// TwinCAT 3 PLC project PLC
// ProgramVersion: 3.1.4024.0
// libraries:
//   Tc2_CncHli, * (Beckhoff Automation GmbH)
//   Tc2_Standard, * (Beckhoff Automation GmbH)
//   Tc2_System, * (Beckhoff Automation GmbH)
//   Tc3_Module, * (Beckhoff Automation GmbH)
//   Triamec EtherCAT Lib, * (Triamec Motion AG)
// project tree:
//   GVLs/ Triamec_GVL.TcGVL
//   / PlcTask.TcTTO
//   POUs/ CNC_Axis.TcPOU, MAIN.TcPOU
// real-time tasks:
//   TASK PlcTask: cycle T#10ms, priority 20, ADS port 350
// I/O:
//   DEVICE Device 1 (EtherCAT), AmsNetId 10.20.34.98.2.1
//     Drive 1 (TSD) [TSD_minFW4.22]
//       modules: Axis 0, Axis 0, Axis 0, Axis 0, Axis 0, Axis 1, Axis 1, Axis 1, Axis 1, Axis 1
// variable links:
//   CNC/Axes/Axis_1 <-> Device 1 (EtherCAT)/Drive 1 (TSD)
//     Inputs/ActualPosition <-> Axis 0/MainInputs/ActualPosition
//     Inputs/ActualVelocity <-> Axis 0/VelocityInputs/ActualVelocity
//     Inputs/MessageId <-> Axis 0/Diagnostic / Digital Inputs/MessageId
//     Inputs/Mode of Operation Display <-> Axis 0/MainInputs/Mode of Operation Display
//     Inputs/PositionError <-> Axis 0/PositionInputs/PositionError
//     Inputs/Status Word <-> Axis 0/MainInputs/Status Word
//     Inputs/TorqueActual <-> Axis 0/TorqueInputs/TorqueActual
//     Inputs/WcState <-> WcState/WcState
//     Outputs/Auxiliary Byte <-> Axis 0/MainOutputs/Auxiliary Byte
//     Outputs/Control Word <-> Axis 0/MainOutputs/Control Word
//     Outputs/Mode of Operation <-> Axis 0/MainOutputs/Mode of Operation
//     Outputs/TargetPosition <-> Axis 0/PositionOutputs/TargetPosition
//     Outputs/TargetTorque <-> Axis 0/TorqueOutputs/TargetTorque
//     Outputs/TargetVelocity <-> Axis 0/VelocityOutputs/TargetVelocity
//   CNC/Axes/Axis_2 <-> Device 1 (EtherCAT)/Drive 1 (TSD)
//     Inputs/ActualPosition <-> Axis 1/MainInputs/ActualPosition
//     Inputs/ActualVelocity <-> Axis 1/VelocityInputs/ActualVelocity
//     Inputs/MessageId <-> Axis 1/Diagnostic / Digital Inputs/MessageId
//     Inputs/Mode of Operation Display <-> Axis 1/MainInputs/Mode of Operation Display
//     Inputs/PositionError <-> Axis 1/PositionInputs/PositionError
//     Inputs/Status Word <-> Axis 1/MainInputs/Status Word
//     Inputs/TorqueActual <-> Axis 1/TorqueInputs/TorqueActual
//     Inputs/WcState <-> WcState/WcState
//     Outputs/Auxiliary Byte <-> Axis 1/MainOutputs/Auxiliary Byte
//     Outputs/Control Word <-> Axis 1/MainOutputs/Control Word
//     Outputs/Mode of Operation <-> Axis 1/MainOutputs/Mode of Operation
//     Outputs/TargetPosition <-> Axis 1/PositionOutputs/TargetPosition
//     Outputs/TargetTorque <-> Axis 1/TorqueOutputs/TargetTorque
//     Outputs/TargetVelocity <-> Axis 1/VelocityOutputs/TargetVelocity

CONFIGURATION PLC
    RESOURCE PLC ON TwinCAT3
        TASK PlcTask(INTERVAL := T#10ms, PRIORITY := 20);
        PROGRAM MAIN WITH PlcTask : MAIN;
    END_RESOURCE
END_CONFIGURATION

// ---- GVLs/Triamec_GVL.TcGVL
VAR_GLOBAL
	gEnableAxes			: BOOL;	(* variable to enable all axes *)
	gStatusAxesEnabled 	: BOOL;	(* variable indicates that all axes enabled *)	
END_VAR

// ---- POUs/MAIN.TcPOU
PROGRAM MAIN
VAR
	Axis		: ARRAY [0..1] OF CNC_Axis; // CNC axis
	Hli 		: MCV_HliInterface;
	axisIdx		: UINT;
END_VAR

(* configuration *)
Axis[0].config.driveId	:= 1001;				// Drive 1 (TSD)/EtherCAT/EtherCAT-Addr.
Axis[0].config.netId	:= '192.168.10.99.2.1';	// Drive 1 (TSD)^InfoData^AdsAddr^netId
Axis[0].config.axisNumber:= 0;					// first (0) or second (1) axis of a dual axis drive
Axis[0].config.axisId	:= 0;					// cnc-axis-id used in events
Axis[1].config.driveId	:= 1001;				// Drive 1 (TSD)/EtherCAT/EtherCAT-Addr.
Axis[1].config.netId	:= '192.168.10.99.2.1';	// Drive 1 (TSD)^InfoData^AdsAddr^netId
Axis[1].config.axisNumber:= 1;					// first (0) or second (1) axis of a dual axis drive
Axis[1].config.axisId	:= 1;					// cnc-axis-id used in events

(* HLI interface *)
IF NOT Hli.Initialized THEN
	Hli(); //initialize HLI
END_IF

(* Axis handler *)
IF Hli.Initialized THEN
	gStatusAxesEnabled := TRUE;
	FOR axisIdx := 0 TO SIZEOF(Axis)/SIZEOF(Axis[0])-1 DO
		Axis[axisIdx].enable := gEnableAxes;
		Axis[axisIdx]();
		IF NOT Axis[axisIdx].enabled THEN
			gStatusAxesEnabled := FALSE;
		END_IF
	END_FOR
END_IF

END_PROGRAM

// ---- POUs/CNC_Axis.TcPOU
FUNCTION_BLOCK CNC_Axis EXTENDS TE_AxisBase0
VAR_INPUT
	enable		: BOOL;
	hold		: BOOL;
END_VAR
VAR_OUTPUT
	ready		: BOOL;
	enabled		: BOOL;
	referenced	: BOOL;
	state		: DWORD;
	error		: BOOL;
END_VAR
VAR
	pAxis		: POINTER TO HIGH_LEVEL_INTERFACE_AX;
END_VAR

(* Triamec Motion AG, 6340 Baar, Switzerland    *)
(* Sample Code may be adapted to customer needs *)
(* -------------------------------------------- *)
(* 
	we do not want any offset between drive and cnc 
    because the drives have there own setPosition
	therefore set the following parameters in the axis of the cnc:
		kenngr.abs_pos_gueltig			1
		kenngr.set_refpos_mode         	OFFSET
		kenngr.set_refpos_offset		0
	this mode ensures, that the cnc does not set cmdPos=actPos when
	MCControlBoolUnit_SetReferencePosition is set
	
	To enable homing using G74 set the following in every axis configuration
	kenngr.device_id  8             ( turn off the target reached check before homing)
*)

IF config.axisId >= 0 AND HLI_SYS_AX_MAXIDX > config.axisId THEN (* check for axis id *)
	(* be careful, array indices start with 0 in TwinCAT 3. Axis starts with 1 *)
	pAxis := gpAx[config.axisId];
	pAxis^.head.plc_present_w := TRUE;
	
	(* enable PLC to drive HLI interface *)
	pAxis^.lr_mc_control.torque_permission.enable_w			:= TRUE;
	pAxis^.lr_mc_control.release_feedhold.enable_w 			:= TRUE;
	pAxis^.lr_mc_control.drive_on.enable_w 					:= TRUE;		
	(* set reference postion offset *)
//	pAxis^.lr_mc_control.set_reference_position.enable_w	:= TRUE;
	(* enable the axis to tracking operation (follow up) *)
	pAxis^.lr_mc_control.follow_up.enable_w 				:= TRUE;

	(* set regulation and feed *)
	pAxis^.lr_mc_control.torque_permission.command_w		:= enable;
	pAxis^.lr_mc_control.release_feedhold.command_w 		:= NOT Hold;
	pAxis^.lr_mc_control.drive_on.command_w 				:= TRUE;
	
	state := pAxis^.lr_state.native_drive_state_r;
	error := (state AND 16#8) <> 0;
	
	(* The axis is set to tracking operation (follow up) on or off, i.e. the control loop is opened.
	   The command position implicitly is set to the actual position. *)
	pAxis^.lr_mc_control.follow_up.command_w				:= (state AND 16#0100) <> 0;
	(* HomingPosition *)
//	pAxis^.lr_mc_control.set_reference_position.command_w	:= (driveState AND 16#8000) <> 0;
	
	ready := pAxis^.lr_state.ready_for_control_loop_on_r;
	enabled := pAxis^.lr_state.ready_for_control_loop_on_r AND pAxis^.lr_state.ready_for_power_on_r AND pAxis^.lr_state.native_drive_state_r.1;
	referenced := pAxis^.lr_state.homing_done_r;
	
END_IF

(* This handles errors (error=TRUE) and warnings (error=FALSE) as TwinCat message *)
CallSlow();

END_FUNCTION_BLOCK
